// TIA Portal V20 export
TYPE "typeCmControlNodeSoftCam"
// stored: Namespace Unit1.Em8
   STRUCT
      thicknessAxisZ : "Unit1.Em8.typeCmControlNodeSoftCamthicknessAxisZ";
   END_STRUCT;
END_TYPE
